TYPE ST_HW_CONTROL_DEV :
STRUCT
	bRotOmronSensor1Feed AT %Q* :BOOL;  // s4: ch1: Feed omron sensor 1
	bRotOmronSensor2Feed AT %Q* :BOOL;  // s4: ch2: Feed omron sensor 2
END_STRUCT
END_TYPE

(* stored: Version 1.1.0.1, ProductVersion 3.1.4024.6
   DUT ST_HW_CONTROL_DEV: Id {3fa93026-3cf8-482e-a913-be8c338af072} *)
